FUNCTION_BLOCK ModbusWriteOutputs
VAR_INPUT
	Data : BYTE;
END_VAR
	
VAR_OUTPUT
	bBUSY : BOOL;
	bError : BOOL;
	nErrId : UDINT;
END_VAR

VAR
	fbwriteoutputs : FB_MBWriteCoils;
END_VAR

fbwriteoutputs(
	sIPAddr := '127.0.0.1', 
	nTCPPort := 505, 
	nUnitID := 255,
	nQuantity := 2,
	nMBAddr := 0, 
	cbLength := SIZEOF(Data),
	pSrcAddr := ADR(Data),
	bExecute := TRUE, 
	tTimeout := T#1S,
);

END_FUNCTION_BLOCK

(* stored: Version 1.1.0.1, ProductVersion 3.1.4024.9
   POU ModbusWriteOutputs: Id {a6f83a06-bd47-44b4-8f92-0c3025a80c44}, SpecialFunc None *)
